KUKA KRL program: STOP.src

&ACCESS RVO1
&COMMENT
DEF STOP(pallet_pick_point:out, ip:out)
decl pos pallet_pick_point
DECL INT ip

;FOLD INI
  ;FOLD BASISTECH INI
    GLOBAL INTERRUPT DECL 3 WHEN $STOPMESS==TRUE DO IR_STOPM ( )
    INTERRUPT ON 3
    BAS (#INITMOV,0 )
  ;ENDFOLD (BASISTECH INI)
  ;FOLD USER INI
    ;Make your modifications here

  ;ENDFOLD (USER INI)
;ENDFOLD (INI)
  BRAKE
  WAIT SEC 0
  HALT
  ip = 1
  pallet_pick_point = $POS_ACT ; remember the actual position to the actual_pick_point_1
END
